KUKA KRL program: ps_2_geo_x1.src, ps_2_geo_x1.dat

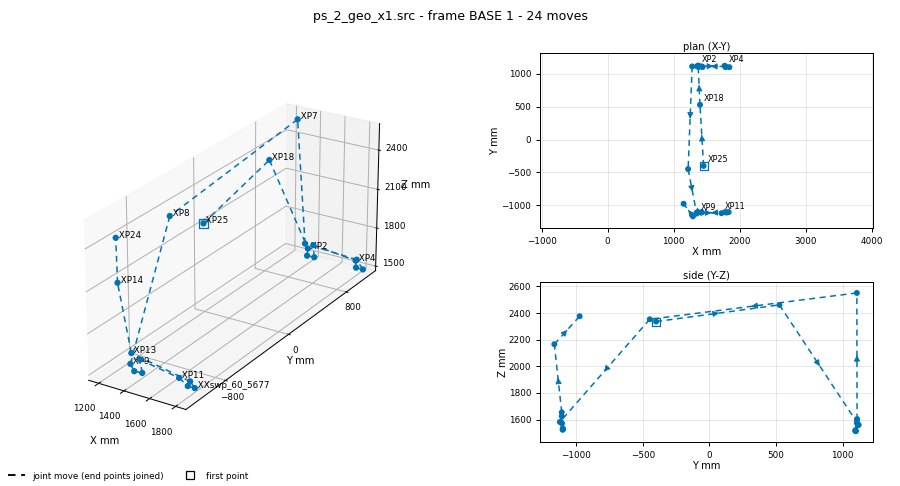
[picture p0: tool path of ps_2_geo_x1.src in frame BASE 1, 24 of 24 moves have a stored position in this frame; points joined in program order, loops and branches not executed]
--- ps_2_geo_x1.src ---
&ACCESS RVO1
&REL 134
&COMMENT SOLDA GUN X1 COM GRIPPER
&PARAM DISKPATH = KRC:\R1\Program
DEF ps_2_geo_x1( )
;FOLD INI
;FOLD SPOTTECH INI
USERSPOT(#INIT)
;ENDFOLD (SPOTTECH INI)
;FOLD GRIPPERTECH INI
USER_GRP(0,DUMMY,DUMMY,GDEFAULT)
;ENDFOLD (GRIPPERTECH INI)
  ;FOLD USER INI
    ;Make your modifications here

  ;ENDFOLD (USER INI)
;ENDFOLD (INI)

; Caracterização dos meios de produção MBB :
; Changes: Solda Geometria Pinca X1 Part2  :
; Modelo: Actros LTA/LTB/MGS/MGSB          :
; Versão Atual: 21/07/2015                 :
; Name: P13.050-R5                         :

chk_w2_wechs_ok ( )      ; CHECK FERRAMENTA: X1

;FOLD OUT 3348 'Fora area GEOBOX' State=FALSE ;%{PE}%R 8.2.20,%MKUKATPBASIS,%COUT,%VOUTX,%P 2:3348, 3:Fora area GEOBOX, 5:FALSE, 6:
$OUT[3348]=FALSE
;ENDFOLD

;FOLD PTP P25 Vel=100 % PDAT35 Tool[2]:Gun X01 Base[1]:ACTROS;%{PE}%R 8.2.20,%MKUKATPBASIS,%CMOVE,%VPTP,%P 1:PTP, 2:P25, 3:, 5:100, 7:PDAT35
$BWDSTART=FALSE
PDAT_ACT=PPDAT35
FDAT_ACT=FP25
BAS(#PTP_PARAMS,100)
PTP XP25
;ENDFOLD
;FOLD PTP P18 CONT Vel=100 % PDAT28 Tool[2]:Gun X01 Base[1]:ACTROS;%{PE}%R 8.2.20,%MKUKATPBASIS,%CMOVE,%VPTP,%P 1:PTP, 2:P18, 3:C_DIS, 5:100, 7:PDAT28
$BWDSTART=FALSE
PDAT_ACT=PPDAT28
FDAT_ACT=FP18
BAS(#PTP_PARAMS,100)
PTP XP18 C_DIS
;ENDFOLD

;FOLD OUT 3339 'R5 aguarda lib soldar geometria' State=TRUE ;%{PE}%R 8.2.20,%MKUKATPBASIS,%COUT,%VOUTX,%P 2:3339, 3:R5 aguarda lib soldar geometria, 5:TRUE, 6:
$OUT[3339]=TRUE
;ENDFOLD
;FOLD WAIT FOR ( IN 3339 'Aguarda lib soldar geometria' );%{PE}%R 8.2.20,%MKUKATPBASIS,%CEXT_WAIT_FOR,%VEXT_WAIT_FOR,%P 2:, 4:, 5:$IN, 6:3339, 7:Aguarda lib soldar geometria, 9:
WAIT FOR  ( $IN[3339] )
;ENDFOLD
;FOLD OUT 3339 'R5 aguarda lib soldar geometria' State=FALSE ;%{PE}%R 8.2.20,%MKUKATPBASIS,%COUT,%VOUTX,%P 2:3339, 3:R5 aguarda lib soldar geometria, 5:FALSE, 6:
$OUT[3339]=FALSE
;ENDFOLD
;FOLD Collision.Monitoring_2_On ;%{PE}%MKUKATPUSER
COLLSTOP( 2, 1 ) ;Interrupt-Controlled
;ENDFOLD
;FOLD ;%{PE}%R 8.2.20,%MKUKATPBASIS,%CCOMMENT,%VNORMAL,%P 2:
;ENDFOLD
;FOLD PTP P2 CONT Vel=100 % PDAT2 Tool[2]:Gun X01 Base[1]:ACTROS;%{PE}%R 8.2.20,%MKUKATPBASIS,%CMOVE,%VPTP,%P 1:PTP, 2:P2, 3:C_DIS, 5:100, 7:PDAT2
$BWDSTART=FALSE
PDAT_ACT=PPDAT2
FDAT_ACT=FP2
BAS(#PTP_PARAMS,100)
PTP XP2 C_DIS
;ENDFOLD

;FOLD ; swp_60_5654;%{PE}%R 8.2.20,%MKUKATPBASIS,%CCOMMENT,%VNORMAL,%P 2:swp_60_5654
;ENDFOLD
;FOLD PTP Xswp_60_5654 PDAT3 SPOT Gun=2 RETR CLS PgNo1=138 ACTIVE=1 Tool[2]:Gun X01 Base[1]:ACTROS;%{PE}%R 8.2.2,%MKUKATPSPOT,%CSPOT,%VPTP,%P 1:PTP, 2:Xswp_60_5654, 3:, 5:100, 7:PDAT3, 10:2, 12:#FIRST, 14:#CLO, 16:189, 18:1, 20:0, 22:0, 24:1, 25:SDAT1
$BWDSTART=FALSE
PDAT_ACT=PPDAT3
FDAT_ACT=FXswp_60_5654
BAS(#PTP_PARAMS,PPDAT3.VEL)
S_ACT.GUN=2
S_ACT.PAIR=SDEFAULT.PAIR
S_ACT.RETR=#CLO
S_ACT.CLO_TM=1
S_ACT.PgNo1=138
S_ACT.PGNO2=SDEFAULT.PGNO2
S_ACT.PRESS1=SDEFAULT.PRESS1
S_ACT.PRESS2=SDEFAULT.PRESS2
S_READY=FALSE
PTP XXswp_60_5654
USERSPOT(#SPOT, S_ACT)
WAIT FOR S_READY
;ENDFOLD

;FOLD ; swp_60_5658;%{PE}%R 8.2.20,%MKUKATPBASIS,%CCOMMENT,%VNORMAL,%P 2:swp_60_5658
;ENDFOLD
;FOLD PTP Xswp_60_5658 PDAT4 SPOT Gun=2 RETR CLS PgNo1=139 ACTIVE=1 Tool[2]:Gun X01 Base[1]:ACTROS;%{PE}%R 8.2.2,%MKUKATPSPOT,%CSPOT,%VPTP,%P 1:PTP, 2:Xswp_60_5658, 3:, 5:100, 7:PDAT4, 10:2, 12:#FIRST, 14:#CLO, 16:190, 18:1, 20:0, 22:0, 24:1, 25:SDAT2
$BWDSTART=FALSE
PDAT_ACT=PPDAT4
FDAT_ACT=FXswp_60_5658
BAS(#PTP_PARAMS,PPDAT4.VEL)
S_ACT.GUN=2
S_ACT.PAIR=SDEFAULT.PAIR
S_ACT.RETR=#CLO
S_ACT.CLO_TM=1
S_ACT.PgNo1=139
S_ACT.PGNO2=SDEFAULT.PGNO2
S_ACT.PRESS1=SDEFAULT.PRESS1
S_ACT.PRESS2=SDEFAULT.PRESS2
S_READY=FALSE
PTP XXswp_60_5658
USERSPOT(#SPOT, S_ACT)
WAIT FOR S_READY
;ENDFOLD

;FOLD PTP P3 CONT Vel=100 % PDAT6 Tool[2]:Gun X01 Base[1]:ACTROS;%{PE}%R 8.2.20,%MKUKATPBASIS,%CMOVE,%VPTP,%P 1:PTP, 2:P3, 3:C_DIS, 5:100, 7:PDAT6
$BWDSTART=FALSE
PDAT_ACT=PPDAT6
FDAT_ACT=FP3
BAS(#PTP_PARAMS,100)
PTP XP3 C_DIS
;ENDFOLD
;FOLD PTP P4 CONT Vel=100 % PDAT7 Tool[2]:Gun X01 Base[1]:ACTROS;%{PE}%R 8.2.20,%MKUKATPBASIS,%CMOVE,%VPTP,%P 1:PTP, 2:P4, 3:C_DIS, 5:100, 7:PDAT7
$BWDSTART=FALSE
PDAT_ACT=PPDAT7
FDAT_ACT=FP4
BAS(#PTP_PARAMS,100)
PTP XP4 C_DIS
;ENDFOLD

;FOLD ; swp_60_5680;%{PE}%R 8.2.20,%MKUKATPBASIS,%CCOMMENT,%VNORMAL,%P 2:swp_60_5680
;ENDFOLD
;FOLD PTP Xswp_60_5680 PDAT8 SPOT Gun=2 RETR CLS PgNo1=140 ACTIVE=1 Tool[2]:Gun X01 Base[1]:ACTROS;%{PE}%R 8.2.2,%MKUKATPSPOT,%CSPOT,%VPTP,%P 1:PTP, 2:Xswp_60_5680, 3:, 5:100, 7:PDAT8, 10:2, 12:#FIRST, 14:#CLO, 16:191, 18:1, 20:0, 22:0, 24:1, 25:SDAT3
$BWDSTART=FALSE
PDAT_ACT=PPDAT8
FDAT_ACT=FXswp_60_5680
BAS(#PTP_PARAMS,PPDAT8.VEL)
S_ACT.GUN=2
S_ACT.PAIR=SDEFAULT.PAIR
S_ACT.RETR=#CLO
S_ACT.CLO_TM=1
S_ACT.PgNo1=140
S_ACT.PGNO2=SDEFAULT.PGNO2
S_ACT.PRESS1=SDEFAULT.PRESS1
S_ACT.PRESS2=SDEFAULT.PRESS2
S_READY=FALSE
PTP XXswp_60_5680
USERSPOT(#SPOT, S_ACT)
WAIT FOR S_READY
;ENDFOLD

;FOLD ; swp_60_5678;%{PE}%R 8.2.20,%MKUKATPBASIS,%CCOMMENT,%VNORMAL,%P 2:swp_60_5678
;ENDFOLD
;FOLD PTP Xswp_60_5678 PDAT9 SPOT Gun=2 RETR CLS PgNo1=141 ACTIVE=1 Tool[2]:Gun X01 Base[1]:ACTROS;%{PE}%R 8.2.2,%MKUKATPSPOT,%CSPOT,%VPTP,%P 1:PTP, 2:Xswp_60_5678, 3:, 5:100, 7:PDAT9, 10:2, 12:#FIRST, 14:#CLO, 16:192, 18:1, 20:0, 22:0, 24:1, 25:SDAT4
$BWDSTART=FALSE
PDAT_ACT=PPDAT9
FDAT_ACT=FXswp_60_5678
BAS(#PTP_PARAMS,PPDAT9.VEL)
S_ACT.GUN=2
S_ACT.PAIR=SDEFAULT.PAIR
S_ACT.RETR=#CLO
S_ACT.CLO_TM=1
S_ACT.PgNo1=141
S_ACT.PGNO2=SDEFAULT.PGNO2
S_ACT.PRESS1=SDEFAULT.PRESS1
S_ACT.PRESS2=SDEFAULT.PRESS2
S_READY=FALSE
PTP XXswp_60_5678
USERSPOT(#SPOT, S_ACT)
WAIT FOR S_READY
;ENDFOLD

;FOLD PTP P5 CONT Vel=100 % PDAT10 Tool[2]:Gun X01 Base[1]:ACTROS;%{PE}%R 8.2.20,%MKUKATPBASIS,%CMOVE,%VPTP,%P 1:PTP, 2:P5, 3:C_DIS, 5:100, 7:PDAT10
$BWDSTART=FALSE
PDAT_ACT=PPDAT10
FDAT_ACT=FP5
BAS(#PTP_PARAMS,100)
PTP XP5 C_DIS
;ENDFOLD
;FOLD PTP P6 CONT Vel=100 % PDAT11 Tool[2]:Gun X01 Base[1]:ACTROS;%{PE}%R 8.2.20,%MKUKATPBASIS,%CMOVE,%VPTP,%P 1:PTP, 2:P6, 3:C_DIS, 5:100, 7:PDAT11
$BWDSTART=FALSE
PDAT_ACT=PPDAT11
FDAT_ACT=FP6
BAS(#PTP_PARAMS,100)
PTP XP6 C_DIS
;ENDFOLD
;FOLD PTP P7 Vel=100 % PDAT12 Tool[2]:Gun X01 Base[1]:ACTROS;%{PE}%R 8.2.20,%MKUKATPBASIS,%CMOVE,%VPTP,%P 1:PTP, 2:P7, 3:, 5:100, 7:PDAT12
$BWDSTART=FALSE
PDAT_ACT=PPDAT12
FDAT_ACT=FP7
BAS(#PTP_PARAMS,100)
PTP XP7
;ENDFOLD
;FOLD  ;%{PE}%R 8.2.20,%MKUKATPBASIS,%CCOMMENT,%VNORMAL,%P 2:
;ENDFOLD
;FOLD Collision.Monitoring_2_Off . ;%{PE}%MKUKATPUSER
COLLSTOP( 2, 2+0 )
;ENDFOLD
;FOLD  ;%{PE}%R 8.2.20,%MKUKATPBASIS,%CCOMMENT,%VNORMAL,%P 2:
;ENDFOLD
;FOLD PTP P8 CONT Vel=100 % PDAT13 Tool[2]:Gun X01 Base[1]:ACTROS;%{PE}%R 8.2.20,%MKUKATPBASIS,%CMOVE,%VPTP,%P 1:PTP, 2:P8, 3:C_DIS, 5:100, 7:PDAT13
$BWDSTART=FALSE
PDAT_ACT=PPDAT13
FDAT_ACT=FP8
BAS(#PTP_PARAMS,100)
PTP XP8 C_DIS
;ENDFOLD
;FOLD  ;%{PE}%R 8.2.20,%MKUKATPBASIS,%CCOMMENT,%VNORMAL,%P 2:
;ENDFOLD
;FOLD Collision.Monitoring_1_On ;%{PE}%MKUKATPUSER
COLLSTOP( 1, 1 ) ;Interrupt-Controlled
;ENDFOLD
;FOLD  ;%{PE}%R 8.2.20,%MKUKATPBASIS,%CCOMMENT,%VNORMAL,%P 2:
;ENDFOLD
;FOLD PTP P9 CONT Vel=100 % PDAT14 Tool[2]:Gun X01 Base[1]:ACTROS;%{PE}%R 8.2.20,%MKUKATPBASIS,%CMOVE,%VPTP,%P 1:PTP, 2:P9, 3:C_DIS, 5:100, 7:PDAT14
$BWDSTART=FALSE
PDAT_ACT=PPDAT14
FDAT_ACT=FP9
BAS(#PTP_PARAMS,100)
PTP XP9 C_DIS
;ENDFOLD

;FOLD ; swp_60_5653;%{PE}%R 8.2.20,%MKUKATPBASIS,%CCOMMENT,%VNORMAL,%P 2:swp_60_5653
;ENDFOLD
;FOLD PTP Xswp_60_5653 PDAT15 SPOT Gun=2 RETR CLS PgNo1=142 ACTIVE=1 Tool[2]:Gun X01 Base[1]:ACTROS;%{PE}%R 8.2.2,%MKUKATPSPOT,%CSPOT,%VPTP,%P 1:PTP, 2:Xswp_60_5653, 3:, 5:100, 7:PDAT15, 10:2, 12:#FIRST, 14:#CLO, 16:193, 18:1, 20:0, 22:0, 24:1, 25:SDAT5
$BWDSTART=FALSE
PDAT_ACT=PPDAT15
FDAT_ACT=FXswp_60_5653
BAS(#PTP_PARAMS,PPDAT15.VEL)
S_ACT.GUN=2
S_ACT.PAIR=SDEFAULT.PAIR
S_ACT.RETR=#CLO
S_ACT.CLO_TM=1
S_ACT.PgNo1=142
S_ACT.PGNO2=SDEFAULT.PGNO2
S_ACT.PRESS1=SDEFAULT.PRESS1
S_ACT.PRESS2=SDEFAULT.PRESS2
S_READY=FALSE
PTP XXswp_60_5653
USERSPOT(#SPOT, S_ACT)
WAIT FOR S_READY
;ENDFOLD

;FOLD ; swp_60_5657;%{PE}%R 8.2.20,%MKUKATPBASIS,%CCOMMENT,%VNORMAL,%P 2:swp_60_5657
;ENDFOLD
;FOLD PTP Xswp_60_5657 PDAT16 SPOT Gun=2 RETR CLS PgNo1=143 ACTIVE=1 Tool[2]:Gun X01 Base[1]:ACTROS;%{PE}%R 8.2.2,%MKUKATPSPOT,%CSPOT,%VPTP,%P 1:PTP, 2:Xswp_60_5657, 3:, 5:100, 7:PDAT16, 10:2, 12:#FIRST, 14:#CLO, 16:194, 18:1, 20:0, 22:0, 24:1, 25:SDAT6
$BWDSTART=FALSE
PDAT_ACT=PPDAT16
FDAT_ACT=FXswp_60_5657
BAS(#PTP_PARAMS,PPDAT16.VEL)
S_ACT.GUN=2
S_ACT.PAIR=SDEFAULT.PAIR
S_ACT.RETR=#CLO
S_ACT.CLO_TM=1
S_ACT.PgNo1=143
S_ACT.PGNO2=SDEFAULT.PGNO2
S_ACT.PRESS1=SDEFAULT.PRESS1
S_ACT.PRESS2=SDEFAULT.PRESS2
S_READY=FALSE
PTP XXswp_60_5657
USERSPOT(#SPOT, S_ACT)
WAIT FOR S_READY
;ENDFOLD

;FOLD PTP P10 CONT Vel=100 % PDAT18 Tool[2]:Gun X01 Base[1]:ACTROS;%{PE}%R 8.2.20,%MKUKATPBASIS,%CMOVE,%VPTP,%P 1:PTP, 2:P10, 3:C_DIS, 5:100, 7:PDAT18
$BWDSTART=FALSE
PDAT_ACT=PPDAT18
FDAT_ACT=FP10
BAS(#PTP_PARAMS,100)
PTP XP10 C_DIS
;ENDFOLD
;FOLD PTP P11 CONT Vel=100 % PDAT19 Tool[2]:Gun X01 Base[1]:ACTROS;%{PE}%R 8.2.20,%MKUKATPBASIS,%CMOVE,%VPTP,%P 1:PTP, 2:P11, 3:C_DIS, 5:100, 7:PDAT19
$BWDSTART=FALSE
PDAT_ACT=PPDAT19
FDAT_ACT=FP11
BAS(#PTP_PARAMS,100)
PTP XP11 C_DIS
;ENDFOLD

;FOLD ; swp_60_5679;%{PE}%R 8.2.20,%MKUKATPBASIS,%CCOMMENT,%VNORMAL,%P 2:swp_60_5679
;ENDFOLD
;FOLD PTP Xswp_60_5679 PDAT20 SPOT Gun=2 RETR CLS PgNo1=144 ACTIVE=1 Tool[2]:Gun X01 Base[1]:ACTROS;%{PE}%R 8.2.2,%MKUKATPSPOT,%CSPOT,%VPTP,%P 1:PTP, 2:Xswp_60_5679, 3:, 5:100, 7:PDAT20, 10:2, 12:#FIRST, 14:#CLO, 16:195, 18:1, 20:0, 22:0, 24:1, 25:SDAT7
$BWDSTART=FALSE
PDAT_ACT=PPDAT20
FDAT_ACT=FXswp_60_5679
BAS(#PTP_PARAMS,PPDAT20.VEL)
S_ACT.GUN=2
S_ACT.PAIR=SDEFAULT.PAIR
S_ACT.RETR=#CLO
S_ACT.CLO_TM=1
S_ACT.PgNo1=144
S_ACT.PGNO2=SDEFAULT.PGNO2
S_ACT.PRESS1=SDEFAULT.PRESS1
S_ACT.PRESS2=SDEFAULT.PRESS2
S_READY=FALSE
PTP XXswp_60_5679
USERSPOT(#SPOT, S_ACT)
WAIT FOR S_READY
;ENDFOLD

;FOLD ; swp_60_5677;%{PE}%R 8.2.20,%MKUKATPBASIS,%CCOMMENT,%VNORMAL,%P 2:swp_60_5677
;ENDFOLD
;FOLD PTP Xswp_60_5677 PDAT21 SPOT Gun=2 RETR OPN PgNo1=145 ACTIVE=1 Tool[2]:Gun X01 Base[1]:ACTROS;%{PE}%R 8.2.2,%MKUKATPSPOT,%CSPOT,%VPTP,%P 1:PTP, 2:Xswp_60_5677, 3:, 5:100, 7:PDAT21, 10:2, 12:#FIRST, 14:#OPN, 16:196, 18:1, 20:0, 22:0, 24:1, 25:SDAT8
$BWDSTART=FALSE
PDAT_ACT=PPDAT21
FDAT_ACT=FXswp_60_5677
BAS(#PTP_PARAMS,PPDAT21.VEL)
S_ACT.GUN=2
S_ACT.PAIR=SDEFAULT.PAIR
S_ACT.RETR=#OPN
S_ACT.CLO_TM=1
S_ACT.PgNo1=145
S_ACT.PGNO2=SDEFAULT.PGNO2
S_ACT.PRESS1=SDEFAULT.PRESS1
S_ACT.PRESS2=SDEFAULT.PRESS2
S_READY=FALSE
PTP XXswp_60_5677
USERSPOT(#SPOT, S_ACT)
WAIT FOR S_READY
;ENDFOLD

;FOLD PTP P12 CONT Vel=100 % PDAT22 Tool[2]:Gun X01 Base[1]:ACTROS;%{PE}%R 8.2.20,%MKUKATPBASIS,%CMOVE,%VPTP,%P 1:PTP, 2:P12, 3:C_DIS, 5:100, 7:PDAT22
$BWDSTART=FALSE
PDAT_ACT=PPDAT22
FDAT_ACT=FP12
BAS(#PTP_PARAMS,100)
PTP XP12 C_DIS
;ENDFOLD
;FOLD PTP P13 CONT Vel=100 % PDAT23 Tool[2]:Gun X01 Base[1]:ACTROS;%{PE}%R 8.2.20,%MKUKATPBASIS,%CMOVE,%VPTP,%P 1:PTP, 2:P13, 3:C_DIS, 5:100, 7:PDAT23
$BWDSTART=FALSE
PDAT_ACT=PPDAT23
FDAT_ACT=FP13
BAS(#PTP_PARAMS,100)
PTP XP13 C_DIS
;ENDFOLD
;FOLD PTP P14 Vel=100 % PDAT24 Tool[2]:Gun X01 Base[1]:ACTROS;%{PE}%R 8.2.20,%MKUKATPBASIS,%CMOVE,%VPTP,%P 1:PTP, 2:P14, 3:, 5:100, 7:PDAT24
$BWDSTART=FALSE
PDAT_ACT=PPDAT24
FDAT_ACT=FP14
BAS(#PTP_PARAMS,100)
PTP XP14
;ENDFOLD
;FOLD  ;%{PE}%R 8.2.20,%MKUKATPBASIS,%CCOMMENT,%VNORMAL,%P 2:
;ENDFOLD
;FOLD Collision.Monitoring_1_Off . ;%{PE}%MKUKATPUSER
COLLSTOP( 1, 2+0 )
;ENDFOLD
;FOLD  ;%{PE}%R 8.2.20,%MKUKATPBASIS,%CCOMMENT,%VNORMAL,%P 2:
;ENDFOLD
;FOLD PTP P24 CONT Vel=100 % PDAT34 Tool[2]:Gun X01 Base[1]:ACTROS;%{PE}%R 8.2.20,%MKUKATPBASIS,%CMOVE,%VPTP,%P 1:PTP, 2:P24, 3:C_DIS, 5:100, 7:PDAT34
$BWDSTART=FALSE
PDAT_ACT=PPDAT34
FDAT_ACT=FP24
BAS(#PTP_PARAMS,100)
PTP XP24 C_DIS
;ENDFOLD

END

--- ps_2_geo_x1.dat ---
&ACCESS RVO1
&REL 134
&COMMENT SOLDA GUN X1 COM GRIPPER
&PARAM DISKPATH = KRC:\R1\Program
DEFDAT  ps_2_geo_x1
;FOLD EXTERNAL DECLARATIONS;%{PE}%MKUKATPBASIS,%CEXT,%VCOMMON,%P
;FOLD GRIPPERTECH EXT
EXT  H50 (INT  :IN,INT  :IN,INT  :IN,GRP_TYP  :IN )
;ENDFOLD (GRIPPERTECH EXT)
;FOLD SPOTTECH EXT
EXT  USERSPOT (S_COMMAND  :IN,SPOT_TYPE  :IN )
;ENDFOLD (SPOTTECH EXT)
;FOLD BASISTECH EXT;%{PE}%MKUKATPBASIS,%CEXT,%VEXT,%P
EXT  BAS (BAS_COMMAND  :IN,REAL  :IN )
DECL INT SUCCESS
;ENDFOLD (BASISTECH EXT)
;FOLD USER EXT;%{E}%MKUKATPUSER,%CEXT,%VEXT,%P
;Make your modifications here

;ENDFOLD (USER EXT)
;ENDFOLD (EXTERNAL DECLARATIONS)

;# ============ START PATH : swp_p13050r5_l_geo_x2 =============
DECL BASIS_SUGG_T LAST_BASIS={POINT1[] "P26                     ",POINT2[] "P26                     ",CP_PARAMS[] "CPDAT0                  ",PTP_PARAMS[] "PDAT36                  ",CONT[] "C_DIS                   ",CP_VEL[] "2.0                     ",PTP_VEL[] "100                     ",SPL_NAME[] "S0                      "}
DECL E6POS XP2={X 1372.56396,Y 1121.151,Z 1559.76099,A -0.000226671793,B 80.0002365,C 89.9995422,S 2,T 11,E1 0.0,E2 0.0,E3 0.0,E4 0.0,E5 0.0,E6 0.0}
DECL FDAT FP2={TOOL_NO 2,BASE_NO 1,IPO_FRAME #BASE,POINT2[] " ",TQ_STATE FALSE}
DECL PDAT PPDAT2={VEL 100.0,ACC 100.0,APO_DIST 100.0,APO_MODE #CDIS}
DECL SPOT_SUGG_T LAST_SPOT={GUN[] "3                       ",RETR_CMD[] "#OPN                    ",CHOISE[] "#FIRST                  ",CLO_TM[] "0                       ",PGNO1[] "1                       ",PRESS1[] "0                       ",PGNO2[] "1                       ",PRESS2[] "0                       ",SPOT_PARAMS[] "SDAT8                   "}
DECL E6POS XXSWP_60_5654={X 1379.349,Y 1099.43604,Z 1512.67102,A -0.00213924609,B 80.0003204,C 89.9978638,S 2,T 11,E1 0.0,E2 0.0,E3 0.0,E4 0.0,E5 0.0,E6 0.0}
DECL FDAT FXswp_60_5654={TOOL_NO 2,BASE_NO 1,IPO_FRAME #BASE,POINT2[] " ",TQ_STATE FALSE}
DECL PDAT PPDAT3={VEL 100.0,ACC 100.0,APO_DIST 100.0}
DECL SPOT_TYPE SSDAT1={GUN 1,PAIR #FIRST,RETR #OPN,CLO_TM 0,PGNO1 1,PRESS1 0.0,PGNO2 0,PRESS2 0.0}
DECL E6POS XXSWP_60_5658={X 1439.85999,Y 1099.03796,Z 1514.74902,A -8.00172329,B 79.9022522,C 82.1200867,S 2,T 11,E1 0.0,E2 0.0,E3 0.0,E4 0.0,E5 0.0,E6 0.0}
DECL FDAT FXswp_60_5658={TOOL_NO 2,BASE_NO 1,IPO_FRAME #BASE,POINT2[] " ",TQ_STATE FALSE}
DECL PDAT PPDAT4={VEL 100.0,ACC 100.0,APO_DIST 100.0}
DECL SPOT_TYPE SSDAT2={GUN 1,PAIR #FIRST,RETR #OPN,CLO_TM 0,PGNO1 1,PRESS1 0.0,PGNO2 0,PRESS2 0.0}
DECL E6POS XP3={X 1424.39294,Y 1109.00696,Z 1603.73804,A -0.00229110499,B 80.001709,C 89.9982986,S 2,T 11,E1 0.0,E2 0.0,E3 0.0,E4 0.0,E5 0.0,E6 0.0}
DECL FDAT FP3={TOOL_NO 2,BASE_NO 1,IPO_FRAME #BASE,POINT2[] " ",TQ_STATE FALSE}
DECL PDAT PPDAT6={VEL 100.0,ACC 100.0,APO_DIST 0.0,APO_MODE #CDIS}
DECL E6POS XP4={X 1773.25305,Y 1117.02405,Z 1561.59204,A 4.50302687E-05,B 51.6748886,C 89.9994736,S 2,T 11,E1 0.0,E2 0.0,E3 0.0,E4 0.0,E5 0.0,E6 0.0}
DECL FDAT FP4={TOOL_NO 2,BASE_NO 1,IPO_FRAME #BASE,POINT2[] " ",TQ_STATE FALSE}
DECL PDAT PPDAT7={VEL 100.0,ACC 100.0,APO_DIST 100.0,APO_MODE #CDIS}
DECL E6POS XP5={X 1787.11401,Y 1107.51404,Z 1574.97998,A 0.000133368405,B 43.2214508,C 90.0008163,S 2,T 11,E1 0.0,E2 0.0,E3 0.0,E4 0.0,E5 0.0,E6 0.0}
DECL FDAT FP5={TOOL_NO 2,BASE_NO 1,IPO_FRAME #BASE,POINT2[] " ",TQ_STATE FALSE}
DECL PDAT PPDAT8={VEL 100.0,ACC 100.0,APO_DIST 100.0}
DECL SPOT_TYPE SSDAT3={GUN 1,PAIR #FIRST,RETR #OPN,CLO_TM 0,PGNO1 1,PRESS1 0.0,PGNO2 0,PRESS2 0.0}
DECL E6POS XXSWP_60_5680={X 1789.53101,Y 1096.005,Z 1517.32495,A -0.789044321,B 51.6700592,C 89.3808823,S 2,T 11,E1 0.0,E2 0.0,E3 0.0,E4 0.0,E5 0.0,E6 0.0}
DECL FDAT FXswp_60_5680={TOOL_NO 2,BASE_NO 1,IPO_FRAME #BASE,POINT2[] " ",TQ_STATE FALSE}
DECL E6POS XXSWP_60_5678={X 1845.76294,Y 1096.51404,Z 1516.75598,A -0.000519223511,B 51.6742516,C 89.9993362,S 2,T 11,E1 0.0,E2 0.0,E3 0.0,E4 0.0,E5 0.0,E6 0.0}
DECL FDAT FXswp_60_5678={TOOL_NO 2,BASE_NO 1,IPO_FRAME #BASE,POINT2[] " ",TQ_STATE FALSE}
DECL PDAT PPDAT9={VEL 100.0,ACC 100.0,APO_DIST 100.0}
DECL SPOT_TYPE SSDAT4={GUN 1,PAIR #FIRST,RETR #OPN,CLO_TM 0,PGNO1 1,PRESS1 0.0,PGNO2 0,PRESS2 0.0}
DECL PDAT PPDAT10={VEL 100.0,ACC 100.0,APO_DIST 0.0,APO_MODE #CDIS}
DECL E6POS XP6={X 1355.12805,Y 1109.03101,Z 1599.82397,A 0.006179458,B 79.9994278,C 90.0059509,S 2,T 11,E1 0.0,E2 0.0,E3 0.0,E4 0.0,E5 0.0,E6 0.0}
DECL FDAT FP6={TOOL_NO 2,BASE_NO 1,IPO_FRAME #BASE,POINT2[] " ",TQ_STATE FALSE}
DECL PDAT PPDAT11={VEL 100.0,ACC 100.0,APO_DIST 100.0,APO_MODE #CDIS}
DECL E6POS XP7={X 1281.677,Y 1107.53003,Z 2551.08203,A 0.0,B 89.9999466,C 89.9999771,S 2,T 43,E1 0.0,E2 0.0,E3 0.0,E4 0.0,E5 0.0,E6 0.0}
DECL FDAT FP7={TOOL_NO 2,BASE_NO 1,IPO_FRAME #BASE,POINT2[] " ",TQ_STATE FALSE}
DECL PDAT PPDAT12={VEL 100.0,ACC 100.0,APO_DIST 100.0,APO_MODE #CDIS}
DECL E6POS XP8={X 1220.53296,Y -447.852997,Z 2353.40601,A -103.035599,B 85.3184509,C 155.2444,S 2,T 3,E1 0.0,E2 0.0,E3 0.0,E4 0.0,E5 0.0,E6 0.0}
DECL FDAT FP8={TOOL_NO 2,BASE_NO 1,IPO_FRAME #BASE,POINT2[] " ",TQ_STATE FALSE}
DECL PDAT PPDAT13={VEL 100.0,ACC 100.0,APO_DIST 100.0,APO_MODE #CDIS}
DECL E6POS XP9={X 1350.23804,Y -1122.651,Z 1581.89502,A 1.263473E-06,B 79.9995728,C -89.9998169,S 2,T 2,E1 0.0,E2 0.0,E3 0.0,E4 0.0,E5 0.0,E6 0.0}
DECL FDAT FP9={TOOL_NO 2,BASE_NO 1,IPO_FRAME #BASE,POINT2[] " ",TQ_STATE FALSE}
DECL PDAT PPDAT14={VEL 100.0,ACC 100.0,APO_DIST 100.0,APO_MODE #CDIS}
DECL E6POS XXSWP_60_5653={X 1365.146,Y -1101.87305,Z 1523.41797,A 4.527071,B 79.9679337,C -85.5410004,S 2,T 2,E1 0.0,E2 0.0,E3 0.0,E4 0.0,E5 0.0,E6 0.0}
DECL FDAT FXswp_60_5653={TOOL_NO 2,BASE_NO 1,IPO_FRAME #BASE,POINT2[] " ",TQ_STATE FALSE}
DECL PDAT PPDAT15={VEL 100.0,ACC 100.0,APO_DIST 100.0}
DECL SPOT_TYPE SSDAT5={GUN 1,PAIR #FIRST,RETR #OPN,CLO_TM 0,PGNO1 1,PRESS1 0.0,PGNO2 0,PRESS2 0.0}
DECL E6POS XXSWP_60_5657={X 1427.34802,Y -1101.11206,Z 1527.14905,A -0.00145211595,B 79.9986115,C -90.0013123,S 2,T 2,E1 0.0,E2 0.0,E3 0.0,E4 0.0,E5 0.0,E6 0.0}
DECL FDAT FXswp_60_5657={TOOL_NO 2,BASE_NO 1,IPO_FRAME #BASE,POINT2[] " ",TQ_STATE FALSE}
DECL PDAT PPDAT16={VEL 100.0,ACC 100.0,APO_DIST 100.0}
DECL SPOT_TYPE SSDAT6={GUN 1,PAIR #FIRST,RETR #OPN,CLO_TM 0,PGNO1 1,PRESS1 0.0,PGNO2 0,PRESS2 0.0}
DECL E6POS XP10={X 1417.23401,Y -1109.00903,Z 1625.34802,A 0.000425354287,B 80.0005493,C -89.9996033,S 2,T 2,E1 0.0,E2 0.0,E3 0.0,E4 0.0,E5 0.0,E6 0.0}
DECL FDAT FP10={TOOL_NO 2,BASE_NO 1,IPO_FRAME #BASE,POINT2[] " ",TQ_STATE FALSE}
DECL PDAT PPDAT18={VEL 100.0,ACC 100.0,APO_DIST 0.0,APO_MODE #CDIS}
DECL E6POS XP11={X 1725.62,Y -1116.44495,Z 1579.84802,A 0.000104248298,B 54.0004311,C -89.9998398,S 2,T 34,E1 0.0,E2 0.0,E3 0.0,E4 0.0,E5 0.0,E6 0.0}
DECL FDAT FP11={TOOL_NO 2,BASE_NO 1,IPO_FRAME #BASE,POINT2[] " ",TQ_STATE FALSE}
DECL PDAT PPDAT19={VEL 100.0,ACC 100.0,APO_DIST 100.0,APO_MODE #CDIS}
DECL E6POS XXSWP_60_5679={X 1780.83496,Y -1099.77795,Z 1528.75598,A -0.000124016893,B 54.0009499,C -90.0000381,S 2,T 34,E1 0.0,E2 0.0,E3 0.0,E4 0.0,E5 0.0,E6 0.0}
DECL FDAT FXswp_60_5679={TOOL_NO 2,BASE_NO 1,IPO_FRAME #BASE,POINT2[] " ",TQ_STATE FALSE}
DECL PDAT PPDAT20={VEL 100.0,ACC 100.0,APO_DIST 100.0}
DECL SPOT_TYPE SSDAT7={GUN 1,PAIR #FIRST,RETR #OPN,CLO_TM 0,PGNO1 1,PRESS1 0.0,PGNO2 0,PRESS2 0.0}
DECL E6POS XXSWP_60_5677={X 1835.16699,Y -1100.29395,Z 1528.89197,A 0.000596353319,B 54.0006104,C -90.0000076,S 2,T 34,E1 0.0,E2 0.0,E3 0.0,E4 0.0,E5 0.0,E6 0.0}
DECL FDAT FXswp_60_5677={TOOL_NO 2,BASE_NO 1,IPO_FRAME #BASE,POINT2[] " ",TQ_STATE FALSE}
DECL PDAT PPDAT21={VEL 100.0,ACC 100.0,APO_DIST 100.0}
DECL SPOT_TYPE SSDAT8={GUN 1,PAIR #FIRST,RETR #OPN,CLO_TM 0,PGNO1 1,PRESS1 0.0,PGNO2 0,PRESS2 0.0}
DECL E6POS XP12={X 1803.677,Y -1107.18506,Z 1572.229,A 0.000519061286,B 54.000679,C -89.9999924,S 2,T 34,E1 0.0,E2 0.0,E3 0.0,E4 0.0,E5 0.0,E6 0.0}
DECL FDAT FP12={TOOL_NO 2,BASE_NO 1,IPO_FRAME #BASE,POINT2[] " ",TQ_STATE FALSE}
DECL PDAT PPDAT22={VEL 100.0,ACC 100.0,APO_DIST 0.0,APO_MODE #CDIS}
DECL E6POS XP13={X 1350.22595,Y -1109.00195,Z 1654.65002,A 0.000663698884,B 80.0001678,C -89.9994431,S 2,T 2,E1 0.0,E2 0.0,E3 0.0,E4 0.0,E5 0.0,E6 0.0}
DECL FDAT FP13={TOOL_NO 2,BASE_NO 1,IPO_FRAME #BASE,POINT2[] " ",TQ_STATE FALSE}
DECL PDAT PPDAT23={VEL 100.0,ACC 100.0,APO_DIST 100.0,APO_MODE #CDIS}
DECL E6POS XP14={X 1293.59705,Y -1164.60706,Z 2165.88306,A -7.0475812,B 79.955719,C -97.7512665,S 2,T 2,E1 0.0,E2 0.0,E3 0.0,E4 0.0,E5 0.0,E6 0.0}
DECL FDAT FP14={TOOL_NO 2,BASE_NO 1,IPO_FRAME #BASE,POINT2[] " ",TQ_STATE FALSE}
DECL PDAT PPDAT24={VEL 100.0,ACC 100.0,APO_DIST 100.0,APO_MODE #CDIS}
DECL PDAT PPDAT28={VEL 100.0,ACC 100.0,APO_DIST 0.0,APO_MODE #CDIS}
DECL E6POS XP18={X 1400.18604,Y 525.832886,Z 2461.27588,A 172.387299,B 85.5420837,C -78.4193573,S 2,T 42,E1 0.0,E2 0.0,E3 0.0,E4 0.0,E5 0.0,E6 0.0}
DECL FDAT FP18={TOOL_NO 2,BASE_NO 1,IPO_FRAME #BASE,POINT2[] " ",TQ_STATE FALSE}
DECL E6POS XP24={X 1152.354,Y -974.318115,Z 2376.229,A 14.2330303,B 49.8189201,C -12.6609898,S 2,T 2,E1 0.0,E2 0.0,E3 0.0,E4 0.0,E5 0.0,E6 0.0}
DECL FDAT FP24={TOOL_NO 2,BASE_NO 1,IPO_FRAME #BASE,POINT2[] " ",TQ_STATE FALSE}
DECL PDAT PPDAT34={VEL 100.0,ACC 100.0,APO_DIST 100.0,APO_MODE #CDIS}
DECL PDAT PPDAT35={VEL 100.0,ACC 100.0,APO_DIST 100.0,APO_MODE #CDIS}
DECL E6POS XP25={X 1455.13196,Y -400.122803,Z 2336.1189,A -17.1097393,B 86.2236862,C -130.626694,S 2,T 3,E1 0.0,E2 0.0,E3 0.0,E4 0.0,E5 0.0,E6 0.0}
DECL FDAT FP25={TOOL_NO 2,BASE_NO 1,IPO_FRAME #BASE,POINT2[] " ",TQ_STATE FALSE}
ENDDAT
